Yaskawa INFORM job: AAA.JBI

/JOB
//NAME AAA
//POS
///NPOS 12,0,0,0,0,0
///TOOL 1
///POSTYPE PULSE
///PULSE
C00000=-51796,131119,96549,2820,-58847,-3321
C00001=-49049,135607,102730,3661,-60453,-4333
C00002=-48629,111887,70554,4134,-52877,-4776
C00003=-48629,111887,70554,4134,-52877,-4776
C00004=-48176,96781,50794,4564,-48514,-5155
C00005=-45258,99227,53950,5575,-49372,-6341
C00006=-45258,99227,53950,5575,-49372,-6341
C00007=-45814,114981,74678,5046,-53978,-5868
C00008=-48629,111887,70554,4134,-52877,-4776
C00009=-48629,111887,70554,4134,-52877,-4776
C00010=-51475,109589,67508,3169,-52059,-3642
C00011=-51796,131119,96549,2820,-58847,-3321
//INST
///DATE 2023/01/13 15:25
///ATTR SC,RW
///GROUP1 RB1
NOP
'Using Motoman MA2010 Base (ta
'rgets wrt base):
'0.0,0.0,0.0,0.0,0.0,0.0
MOVC C00000 V=20.0 PL=1
MOVC C00001 V=20.0 PL=1
MOVC C00002 V=20.0 PL=0 FPT
MOVC C00003 V=10.0 PL=1
MOVC C00004 V=10.0 PL=1
MOVC C00005 V=10.0 PL=0 FPT
MOVC C00006 V=10.0 PL=1
MOVC C00007 V=10.0 PL=1
MOVC C00008 V=10.0 PL=0 FPT
MOVC C00009 V=10.0 PL=1
MOVC C00010 V=10.0 PL=1
MOVC C00011 V=10.0 PL=0 FPT
END
